RoboDK station: kr30 cnc 090719 3.rdk

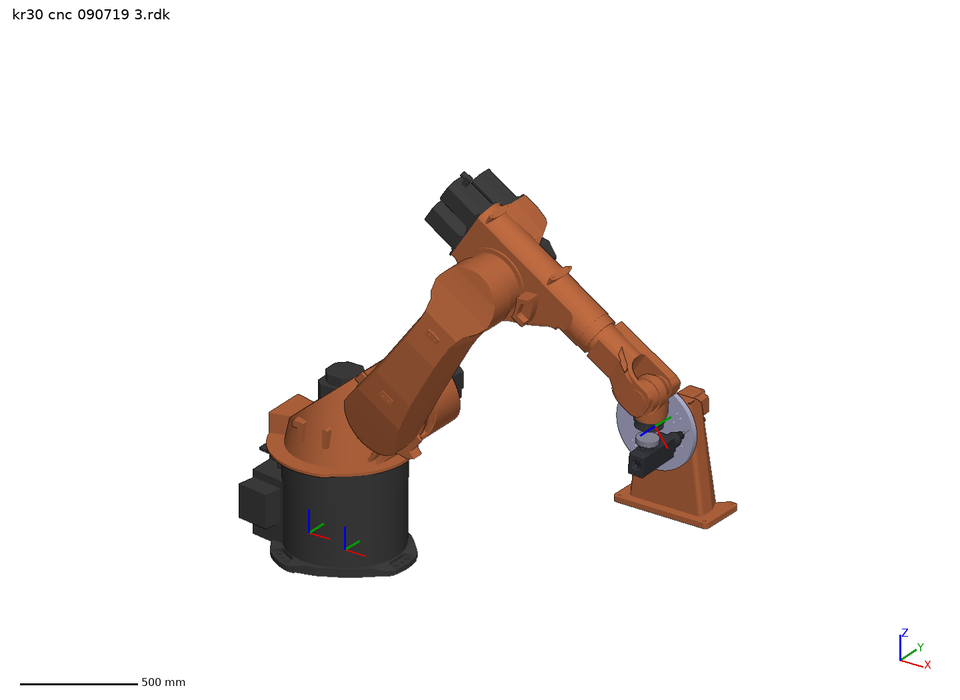
[picture v0: the station drawn from its stored meshes, robots at their saved joint values, targets as dots, program paths as lines]
Station kr30 cnc 090719 3. Poses are relative to the parent item; angles as X-Y-Z fixed-axis rotations.
  - frame GIGASHEEN 7th Axis Base at (-220, 48.2, 0) mm
    - robot KUKA KP1 MD250: 1 axes, payload 250 kg
        modified DH rows (alpha deg, a mm, theta deg, d mm): 0, 0, 0, 0
        base shift (1587.22, 296.05, 828) mm, rotated rx 0 ry 90 rz -90 deg
        joint limits [-3600] to [3600]; home [0]; saved at [1119.52]
      - frame Turntable Base at (0, 0, 0) mm
  - frame GIGASHEEN Base at (0, 0, 0) mm
    - robot GIGASHEEN (model KUKA KR 30 HA): 6 axes, payload 30 kg, reach 2033 mm, repeatability 0.05 mm, weight 665 kg
        modified DH rows (alpha deg, a mm, theta deg, d mm): 0, 0, 0, 815; -90, 350, 0, 0; 0, 850, -90, 0; -90, 145, 0, 820; 90, 0, 0, 0; -90, 0, 180, 170
        joint limits [-185, -135, -120, -350, -119, -350] to [185, 35, 158, 350, 119, 350]; home [0, -90, 90, 0, 0, 0]; saved at [-0.263, -56.336, 89.398, 180.183, -62.071, -268.099]
      - tool 1/2" End Mill TCP, TCP at (338.07, -0.2, 160.37) mm, rotated rx 0 ry 90 rz 0 deg, size 415.8 x 102 x 153.6 mm, geometry from GIGASHEEN
